(* CODESYS project MotionSelector.xml

Project tree, tasks and I/O mapping:
  function block MotionSelector [LD]
*)

// MotionSelector
FUNCTION_BLOCK MotionSelector
VAR_INPUT
	FirstAdvance: BOOL;
	FirstRetract: BOOL;
	RetryAdvance: BOOL;
	RetryRetract: BOOL;
	TearBag: BOOL;
	ResetBag: BOOL;
	RetractOneBag: BOOL;
	BaggerSettings: BaggerSettings;
END_VAR
VAR_OUTPUT
	Execute: BOOL;
	Steps: UDINT;
	Direction: UINT;
	Speed: UINT;
	TriggerOnSensor: BOOL;
END_VAR
VAR
	TOF_0: TOF;
	TON_0: TON;
END_VAR
VAR // added by the converter: edge detectors and wires of the graphical bodies
    _rt1, _rt2, _rt3, _rt4, _rt5, _rt6, _rt7 : R_TRIG;
END_VAR

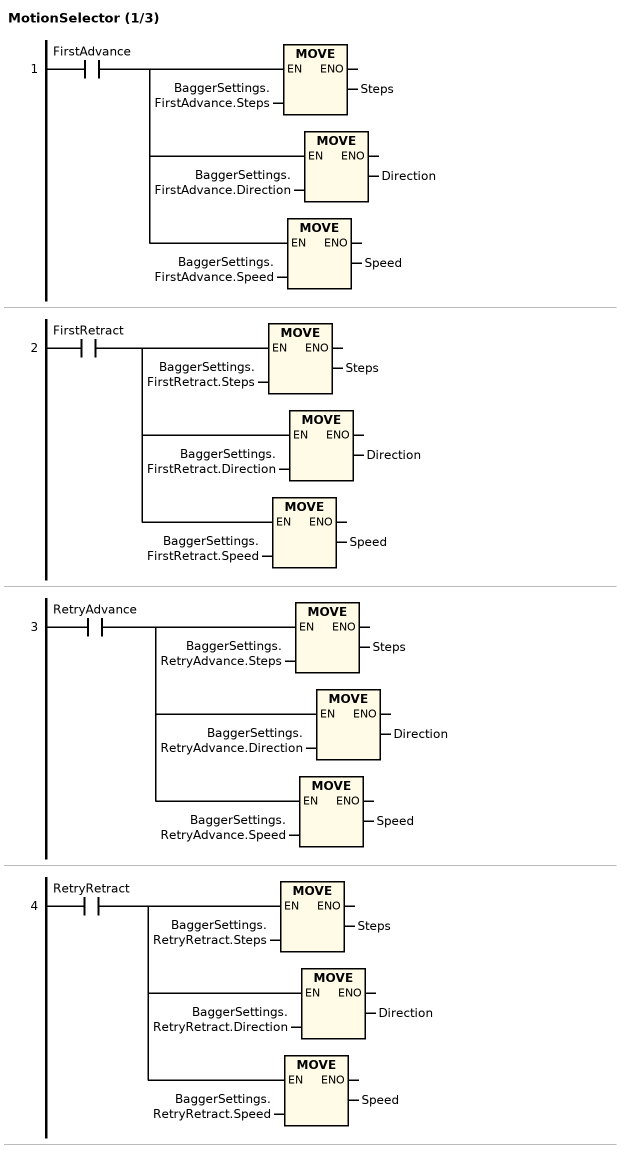
// NETWORK 1
IF FirstAdvance THEN Steps := BaggerSettings.FirstAdvance.Steps; END_IF
IF FirstAdvance THEN Direction := BaggerSettings.FirstAdvance.Direction; END_IF
IF FirstAdvance THEN Speed := BaggerSettings.FirstAdvance.Speed; END_IF

// NETWORK 2
IF FirstRetract THEN Steps := BaggerSettings.FirstRetract.Steps; END_IF
IF FirstRetract THEN Direction := BaggerSettings.FirstRetract.Direction; END_IF
IF FirstRetract THEN Speed := BaggerSettings.FirstRetract.Speed; END_IF

// NETWORK 3
IF RetryAdvance THEN Steps := BaggerSettings.RetryAdvance.Steps; END_IF
IF RetryAdvance THEN Direction := BaggerSettings.RetryAdvance.Direction; END_IF
IF RetryAdvance THEN Speed := BaggerSettings.RetryAdvance.Speed; END_IF

// NETWORK 4
IF RetryRetract THEN Steps := BaggerSettings.RetryRetract.Steps; END_IF
IF RetryRetract THEN Direction := BaggerSettings.RetryRetract.Direction; END_IF
IF RetryRetract THEN Speed := BaggerSettings.RetryRetract.Speed; END_IF

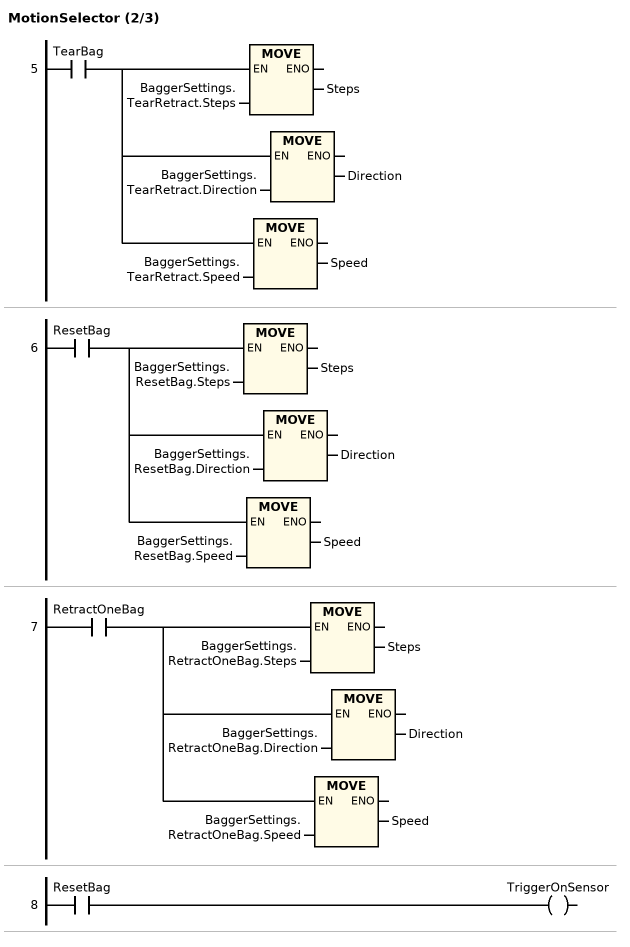
// NETWORK 5
IF TearBag THEN Steps := BaggerSettings.TearRetract.Steps; END_IF
IF TearBag THEN Direction := BaggerSettings.TearRetract.Direction; END_IF
IF TearBag THEN Speed := BaggerSettings.TearRetract.Speed; END_IF

// NETWORK 6
IF ResetBag THEN Steps := BaggerSettings.ResetBag.Steps; END_IF
IF ResetBag THEN Direction := BaggerSettings.ResetBag.Direction; END_IF
IF ResetBag THEN Speed := BaggerSettings.ResetBag.Speed; END_IF

// NETWORK 7
IF RetractOneBag THEN Steps := BaggerSettings.RetractOneBag.Steps; END_IF
IF RetractOneBag THEN Direction := BaggerSettings.RetractOneBag.Direction; END_IF
IF RetractOneBag THEN Speed := BaggerSettings.RetractOneBag.Speed; END_IF

// NETWORK 8
TriggerOnSensor := ResetBag;

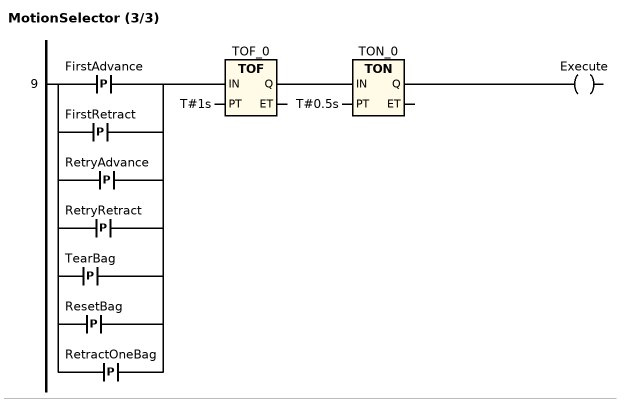
// NETWORK 9
_rt1(CLK := FirstAdvance);
_rt2(CLK := FirstRetract);
_rt3(CLK := RetryAdvance);
_rt4(CLK := RetryRetract);
_rt5(CLK := TearBag);
_rt6(CLK := ResetBag);
_rt7(CLK := RetractOneBag);
TOF_0(IN := _rt1.Q OR _rt2.Q OR _rt3.Q OR _rt4.Q OR _rt5.Q OR _rt6.Q OR _rt7.Q, PT := T#1s); // TOF
TON_0(IN := TOF_0.Q, PT := T#0.5s); // TON
Execute := TON_0.Q;

END_FUNCTION_BLOCK
